// Re-execution, for someone at a keyboard. Separate because it is a debugging
// surface, not something CI or the sequencer should hold.
INTERFACE I_TestReRun EXTENDS __SYSTEM.IQueryInterface

// Re-execute every registered test. Clears verdicts and counts and produces a
// fresh result document.
METHOD ReRun
END_METHOD

// Re-execute one test by label. Records no result and writes no document, so a
// session at the keyboard cannot pollute the CI artifact with duplicate entries.
//
// Returns FALSE if the label is not registered.
METHOD ReRunSingle : BOOL
VAR_INPUT
	Label : T_MaxString;
END_VAR
END_METHOD

END_INTERFACE

(* stored: Version 1.1.0.1
   Itf I_TestReRun: Id {1385606b-00d9-4d3e-ad83-cdee06683859}
   Method ReRun: Id {bc1dce0c-9b26-4ad7-94fc-aa6fd89fe267}
   Method ReRunSingle: Id {ae578273-24f0-4128-9233-5f3a17706219} *)
